// TIA Portal V17 export
// export: Created 2024-08-09T12:53:05.2064458Z, ExportSetting WithDefaults, DisplayName Totally Integrated Automation Portal, DisplayVersion V17 Update 7, DisplayName TIA Portal Openness, DisplayVersion V17 Update 7, DisplayName TIA Portal Version Control Interface, DisplayVersion V17, DisplayName STEP 7 Professional, DisplayVersion V17 Update 7, DisplayName STEP 7 Safety, DisplayVersion V17 Update 6, DisplayName WinCC Professional, DisplayVersion V17 Update 7
VAR_GLOBAL   // PLC tag table "Temporisation"
END_VAR
VAR_GLOBAL CONSTANT   // user constants
   TpFPm : Time := T#30s;   // Temporisation de filtrage de perte du passage matiere du transporteur pour l'acquit fosse vide
   TpPresPm : Time := T#2s;   // Temporisation de filtrage pour prise en compte du passage matiere par l'automatisme
   TpDefPm : Time := T#15s;   // Temporisation d'attente du passage matière avant activation d'un dialogue de défaut
   TpMaskNh : Time := T#25s;   // Temporisation pour masquer le niveau haut
   TpDefNh : Time := T#15s;   // Temporisation pour afficher defaut niveau haut
   TpAvRedAmo : Time := T#10s;   // Temporisation avant redemarage de l'amont
   TpAvArrMobi : Time := T#30s;   // Temporisation avant arret mobile
   TpAvSuspAmo : Time := T#10s;   // Temporisation avant arret amont
   TpAvRedMob : Time := T#20s;   // Temporisation avant redemarage mobile
   TpDefNb : Time := T#15s;   // Temporisation pour afficher defaut niveau bas
END_VAR
